FUNCTION_BLOCK Assembly_LAT

VAR_INPUT
	iSafetyOK			: BOOL := TRUE;
	iPowerOn			: BOOL;
	cmdDivertRight 		: BOOL;
	cmdDivertLeft 		: BOOL;
	cmdPassThru 		: BOOL;
	cmdReceiveRight 	: BOOL;
	cmdReceiveLeft 		: BOOL;
END_VAR

VAR_OUTPUT
	stsIdle				: BOOL;
	stsDivertingRight 	: BOOL;
	stsDivertingLeft 	: BOOL;
	stsPassingThru 		: BOOL;
	stsReceivingRight	: BOOL;
	stsRecevingLeft 	: BOOL;
	stsFaulted 			: BOOL;
	stsFaultCode 		: INT;
END_VAR

VAR_IN_OUT
	PartSensor 			: Device_PartSensor;
	Lift 				: Device_Actuator;
	Transfer			: Device_Motor_OnOff;
END_VAR

VAR
END_VAR

//Map SafetyOK input to Lift and Conv

Lift.iSafetyOK 	:= inpSafetyOK;
Conv.inpSafetyOK 	:= inpSafetyOK;

//Map PowerOn input to Lift and Conv

Lift.iPowerOn 	:= inpPowerOn;
Conv.inpPowerOn 	:= inpPowerOn;

IF PartSensor.oPartPresent THEN
	//Lift.cmdExtend 	:= 1;
	//Conv.cmdRunFwd 	:= 1;
END_IF

END_FUNCTION_BLOCK

(* stored: Version 1.1.0.1, ProductVersion 3.1.4022.11
   POU Assembly_LAT: Id {a0545ff5-c5d0-4f16-8eeb-954c14055efb}, SpecialFunc None *)
